TYPE MoveState_t :
(
	MOVESTATE_INIT,
	MOVESTATE_ENABLE,
	MOVESTATE_FORWARD,
	MOVESTATE_BACKWARDS,
	MOVESTATE_BACKWARDSSLOW,
	MOVESTATE_NEWTARGETPOSITION,
	MOVESTATE_ERROR,
	MOVESTATE_RESET
) UDINT;
END_TYPE

(* stored: Version 1.1.0.1
   DUT MoveState_t: Id {c4f23ecc-e73b-4cde-aa65-84b797479e28} *)
